SUBAPPLICATION T_FF_ILOCK_EVENT (* Toggle-Flip-Flop mit externem RESET-Eingang und SET-Ausgang zur wechselseitigen Verriegelung per Event-Verdrahtung (Radio-Button-Logik). Generisch fuer beliebig viele Teilnehmer verkettbar, indem SET des einen an RESET des naechsten angeschlossen wird. *)
  (* Standard: 61499-2 *)
  (* Version 1.0, 2026-09-09, Franz Höpfinger, Meisterschulen am Ostbahnhof, Ausgelagert aus Uebung_004b3b_sub zur Wiederverwendung fuer weitere verriegelte Toggle-Ketten. *)
  PACKAGE MyLib::sys;
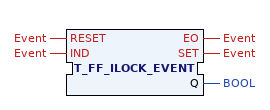
  EVENT_INPUT
    RESET;
    IND;
  END_EVENT
  EVENT_OUTPUT
    EO;
    SET;
  END_EVENT
  VAR_OUTPUT
    Q : BOOL;
  END_VAR
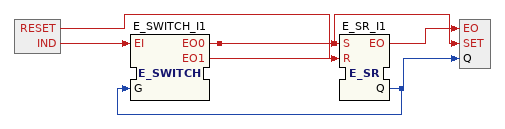
  FBS
    E_SR_I1 : iec61499::events::E_SR;
    E_SWITCH_I1 : iec61499::events::E_SWITCH;
  END_FBS
  EVENT_CONNECTIONS
    E_SWITCH_I1.EO0 TO E_SR_I1.S;
    E_SWITCH_I1.EO1 TO E_SR_I1.R;
    RESET TO E_SR_I1.R;
    E_SR_I1.EO TO EO;
    IND TO E_SWITCH_I1.EI;
    E_SWITCH_I1.EO0 TO SET;
  END_CONNECTIONS
  DATA_CONNECTIONS
    E_SR_I1.Q TO E_SWITCH_I1.G;
    E_SR_I1.Q TO Q;
  END_CONNECTIONS
END_SUBAPPLICATION
